// TwinCAT 3 PLC project plc
// ProgramVersion: 3.1.4024.0
// libraries:
//   Tc2_Standard, * (Beckhoff Automation GmbH)
//   Tc2_System, * (Beckhoff Automation GmbH)
//   Tc3_Module, * (Beckhoff Automation GmbH)
// project tree:
//   DUTs/ PositionAxis.TcDUT, PositionAxis_Status.TcDUT
//   / PlcTask.TcTTO
//   POUs/ MAIN.TcPOU
// real-time tasks:
//   TASK PlcTask: cycle T#2ms, priority 4, ADS port 352
// I/O:
//   DEVICE Device 3 (EtherCAT), AmsNetId 169.254.115.184.4.1
//     Drive 1 (ZeroErr Driver) [ZeroErr Driver]
//     Drive 2 (ZeroErr Driver) [ZeroErr Driver]
//     Drive 3 (ZeroErr Driver) [ZeroErr Driver]
// variable links:
//   plc/plc Instance <-> Device 3 (EtherCAT)/Drive 1 (ZeroErr Driver)
//     PlcTask Inputs/MAIN.P_Axis_1_STATUS/POSITION_VALUE <-> Transmit PDO mapping 0/Position actual value
//     PlcTask Inputs/MAIN.P_Axis_1_STATUS/STATUS_WORD <-> Transmit PDO mapping 0/Status word
//     PlcTask Outputs/MAIN.P_Axis_1_COMMAND/CONTROL_WORD <-> Receive PDO mapping 7/Control word
//     PlcTask Outputs/MAIN.P_Axis_1_COMMAND/MODE_OF_OPERATION <-> Receive PDO mapping 7/Mode of operation
//     PlcTask Outputs/MAIN.P_Axis_1_COMMAND/TARGET_POSIION <-> Receive PDO mapping 7/Target Position
//   plc/plc Instance <-> Device 3 (EtherCAT)/Drive 2 (ZeroErr Driver)
//     PlcTask Inputs/MAIN.P_Axis_2_STATUS/POSITION_VALUE <-> Transmit PDO mapping 0/Position actual value
//     PlcTask Inputs/MAIN.P_Axis_2_STATUS/STATUS_WORD <-> Transmit PDO mapping 0/Status word
//     PlcTask Outputs/MAIN.P_Axis_2_COMMAND/CONTROL_WORD <-> Receive PDO mapping 7/Control word
//     PlcTask Outputs/MAIN.P_Axis_2_COMMAND/MODE_OF_OPERATION <-> Receive PDO mapping 7/Mode of operation
//     PlcTask Outputs/MAIN.P_Axis_2_COMMAND/TARGET_POSIION <-> Receive PDO mapping 7/Target Position

CONFIGURATION plc
    RESOURCE PLC ON TwinCAT3
        TASK PlcTask(INTERVAL := T#1ms, PRIORITY := 4);
        PROGRAM MAIN WITH PlcTask : MAIN;
    END_RESOURCE
END_CONFIGURATION

// ---- DUTs/PositionAxis.TcDUT
TYPE PositionAxis :
STRUCT
	CONTROL_WORD :UINT;
	TARGET_POSIION:DINT;
	MODE_OF_OPERATION:SINT:=1;
END_STRUCT
END_TYPE

// ---- DUTs/PositionAxis_Status.TcDUT
TYPE PositionAxis_Status :
STRUCT
	STATUS_WORD:UINT;
	POSITION_VALUE:DINT;
END_STRUCT
END_TYPE

// ---- POUs/MAIN.TcPOU
PROGRAM MAIN
VAR
	Grap_PositionAxis1 AT%QD100 :PositionAxis;
	Grap_PositionAxis1_Status AT%ID100:PositionAxis_Status;
END_VAR

END_PROGRAM
